Fanuc KAREL source: MP0009.KL

PROGRAM MP0009
%STACKSIZE=65535
%PRIORITY=65535
%NOLOCKGROUP
ROUTINE FINT(P1 : INTEGER) : INTEGER FROM MP0009
ROUTINE FREAL(P1 : REAL) : REAL FROM MP0009
ROUTINE RTEST(P1 : INTEGER; P2 : REAL) FROM MP0009
ROUTINE FINT
BEGIN
-- UNRESOLVED_PC line 5 opcodes [2D 9D 52 7F] marker_code=1
-- UNRESOLVED_PC line 6 opcodes [7F] marker_code=18
END FINT
ROUTINE FREAL
BEGIN
-- UNRESOLVED_PC line 9 opcodes [2D 2E 69 7F] marker_code=28
-- UNRESOLVED_PC line 10 opcodes [7F] marker_code=49
END FREAL
ROUTINE RTEST
VAR
S1 : INTEGER
S2 : INTEGER
U2C_3 : INTEGER -- ASSUMED 2C source type; see uncertainty report
U2C_4 : INTEGER -- ASSUMED 2C source type; see uncertainty report
U2C_5 : INTEGER -- ASSUMED 2C source type; see uncertainty report
U2C_6 : INTEGER -- ASSUMED 2C source type; see uncertainty report
S3 : INTEGER
U2C_8 : REAL -- ASSUMED 2C source type; see uncertainty report
BEGIN
S1=7
S2=3
U2C_3=2
U2C_4=1075838976
U2C_5=1083179008
U2C_6=1069547520
S3=(S1 - S2)
END RTEST
BEGIN
RTEST(7,2.5)
END MP0009
